TYPE SmokeControlStatus :
STRUCT
	Gateway: STRING;
	Device1: STRING;
	Device2: STRING;
	Device3: STRING;
	Device4: STRING;
END_STRUCT
END_TYPE

(* stored: Version 1.1.0.1, ProductVersion 3.1.4024.6
   DUT SmokeControlStatus: Id {ec7a68e3-6dd1-4172-a4c7-a4b57ae8fa8d} *)
